FUNCTION WRITE_PROTECTED_LWORD
VAR_INPUT
    Ptr : POINTER TO LWORD;
    Value : LWORD;
END_VAR

Ptr^ := Value;

END_FUNCTION

(* stored: Version 1.1.0.1, ProductVersion 3.1.4022.18
   POU WRITE_PROTECTED_LWORD: Id {c5f11757-2c55-43b4-9c4e-9a39fdf2cd53}, SpecialFunc None *)
